Universal Robots URScript: a_full_bow_2_27.script

def a_full_bow():
  global _hidden_verificationVariable=0
  step_count_db132347_31d2_4545_98c6_f20b54240faf = 0.0
  thread Step_Counter_Thread_fb8ca14a_9a38_40f6_a6b0_7cbd58039a9b():
    while (True):
      step_count_db132347_31d2_4545_98c6_f20b54240faf = step_count_db132347_31d2_4545_98c6_f20b54240faf + 1.0
      sync()
    end
  end
  run Step_Counter_Thread_fb8ca14a_9a38_40f6_a6b0_7cbd58039a9b()
  set_tcp(p[0.028210348281514253,-0.09610723587300697,-0.09969041498611403,0.0,0.0,0.0])
  set_standard_analog_input_domain(0, 1)
  set_standard_analog_input_domain(1, 1)
  set_tool_analog_input_domain(0, 1)
  set_tool_analog_input_domain(1, 1)
  set_analog_outputdomain(0, 0)
  set_analog_outputdomain(1, 0)
  set_input_actions_to_default()
  set_tool_communication(False, 115200, 0, 1, 1.5, 3.5)
  set_tool_output_mode(0)
  set_tool_digital_output_mode(0, 1)
  set_tool_digital_output_mode(1, 1)
  set_tool_voltage(0)
  set_target_payload(0.260000, [0.050000, -0.008000, 0.024000], [0.000163, 0.000163, 0.000163, 0.000000, 0.000000, 0.000000])
  set_safety_mode_transition_hardness(1)
  set_gravity([0.0, 0.0, 9.82])
  global Plane_1=p[0.32571614183608727,0.7933870146316717,0.11820742021636722,-2.208244884171713,-0.24738609815952348,-1.9195085473101943]
  global Plane_2=p[0.3436052139151623,0.7478032414335104,0.10077839665899768,2.768545736097797,0.1284831553507919,1.3672805628273381]
  global Plane_3=p[0.31945151854627996,0.6757990361168175,0.09459088830114093,2.7301760593116526,-0.049483824131046385,1.4252239353300047]
  global Plane_4=p[0.3372257363094211,0.6222230974198586,0.07001667903587716,2.621672423508307,-0.12240385890263918,1.4373011913128484]
  # begin: URCap Installation Node
  #   Source: External Control, 1.0.5, FZI Research Center for Information Technology
  #   Type: External Control
  # end: URCap Installation Node
  global timer_1=0
  global Waypoint_1_p=p[.300717266074, .793568239540, .099710283103, -1.543522183454, -2.354885618328, 1.346770272474]
  global Waypoint_1_q=[-2.181615177785055, -0.1340765518001099, 0.3750680128680628, -0.918654815559723, -1.5732234160052698, -2.5891388098346155]
  global Waypoint_2_p=p[.473129539189, .413197423330, .256308427905, -1.460522581833, -2.310115543652, 1.445803824327]
  global Waypoint_2_q=[-2.708285633717672, -0.8578118842891236, 1.4135482946978968, -1.2191530925086518, -1.9905441443072718, -2.942223135625021]
  global timer_1_is_counting=False
  thread Timer_Thread():
    while (True):
      if (timer_1_is_counting):
        timer_1 = timer_1 + get_steptime()
      end
      sync()
    end
  end
  run Timer_Thread()
  while (True):
    $ 2 "Robot Program"
    $ 9 "MoveL"
    $ 10 "Waypoint_1" "breakAfter"
    movel(Waypoint_1_p, a=1.2, v=0.25)
    $ 11 "Waypoint_2" "breakAfter"
    movel(Waypoint_2_p, a=1.2, v=0.25)
    $ 12 "MoveL"
    $ 13 "Waypoint_2" "breakAfter"
    movel(Waypoint_2_p, a=1.2, v=0.25)
    $ 14 "Waypoint_1" "breakAfter"
    movel(Waypoint_1_p, a=1.2, v=0.25)
    $ 15 "Wait: 300.0"
    sleep(300.0)
    $ 16 "bow_dir≔ True "
    global bow_dir=  True
    $ 17 "note_dur≔3"
    global note_dur=3
    $ 18 "timer_1: Start"
    timer_1_is_counting = True
    $ 19 "If bow_dir"
    if (bow_dir):
      $ 20 "MoveL"
      $ 21 "Waypoint_2" "breakAfter"
      global move_thread_flag_21=0
      thread move_thread_21():
        enter_critical
        move_thread_flag_21 = 1
        movel(Waypoint_2_p, a=1.2, v=0.25)
        move_thread_flag_21 = 2
        exit_critical
      end
      move_thread_flag_21 = 0
      move_thread_han_21 = run move_thread_21()
      while (True):
        if (timer_1 == note_dur):
          kill move_thread_han_21
          stopl(1.2)
          $ 22 "Until (expression)"
          break
        end
        sleep(1.0E-10)
        if (move_thread_flag_21 > 1):
          join move_thread_han_21
          break
        end
        sync()
      end
    else:
      $ 23 "Else" "noBreak"
      $ 24 "MoveL"
      $ 25 "Waypoint_1" "breakAfter"
      global move_thread_flag_25=0
      thread move_thread_25():
        enter_critical
        move_thread_flag_25 = 1
        movel(Waypoint_1_p, a=1.2, v=0.25)
        move_thread_flag_25 = 2
        exit_critical
      end
      move_thread_flag_25 = 0
      move_thread_han_25 = run move_thread_25()
      while (True):
        if (timer_1 == note_dur):
          kill move_thread_han_25
          stopl(1.2)
          $ 26 "Until (expression)"
          break
        end
        sleep(1.0E-10)
        if (move_thread_flag_25 > 1):
          join move_thread_han_25
          break
        end
        sync()
      end
    end
    $ 31 "timer_1: Stop"
    timer_1_is_counting = False
    $ 32 "timer_1: Reset"
    timer_1 = 0
  end
end
